INTERFACE I_Contents EXTENDS I_Serializable

METHOD PUBLIC GetEnumerator : I_ForwardEnumerator
VAR_INPUT
END_VAR
END_METHOD

METHOD PUBLIC TryGetByName : BOOL
VAR_INPUT
	Name : STRING;
	Destination : REFERENCE TO I_Content;
END_VAR
END_METHOD

END_INTERFACE

(* stored: Version 1.1.0.1, ProductVersion 3.1.4024.12
   Itf I_Contents: Id {fbdd14bf-6b91-0766-32ee-461417efff91}
   Method GetEnumerator: Id {db852c70-8a39-07a6-2dbb-1cd0af417ff2}
   Method TryGetByName: Id {4da7ab31-0944-09cf-2fa6-97fd1ac99ee7} *)
